{attribute addProperty BoxType "EL9227-4433-0018"}
{attribute addProperty Id "OCP_Inputs_ChannelAT %I*ARRAY[0..5] OF OCP_Inputs_Channel_8753EDC6192240OCP_Outputs_ChannelAT %Q*ARRAY[0..1] OF OCP_Outputs_Channel_F330A9163240WcStateAT %I*WcState_98A4DF7520.250InfoDataAT %I*InfoData_BC63D37F80100"}
{attribute addProperty CRC "3994657699"}
{attribute addProperty SizeInBites "306"}
{attribute addProperty SizeInBytes "38.25"}
TYPE EL9227_9D6FA8BB :
STRUCT
	{attribute addProperty Name "OCP_Inputs_Channel"}
	OCP_Inputs_Channel : ARRAY[0..5] OF OCP_Inputs_Channel_8753EDC6;
	{attribute addProperty Name "OCP_Outputs_Channel"}
	OCP_Outputs_Channel : ARRAY[0..1] OF OCP_Outputs_Channel_F330A916;
	{attribute addProperty Name "WcState"}
	WcState : WcState_98A4DF75;
	{attribute addProperty Name "InfoData"}
	InfoData : InfoData_BC63D37F;
END_STRUCT
END_TYPE

(* stored: Version 1.2.0.0, ProductVersion 3.1.4024.9
   DUT EL9227_9D6FA8BB: Id {79101dbb-9f67-4c1d-a419-d1b66908cd3e} *)
